SUBAPPLICATION MF (* Subapplication Type *)
  (* Standard: 61499-2 *)
  (* Version 1.0, 2025-02-12, franz *)
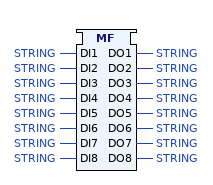
  VAR_INPUT
    DI1 : STRING;
    DI2 : STRING;
    DI3 : STRING;
    DI4 : STRING;
    DI5 : STRING;
    DI6 : STRING;
    DI7 : STRING;
    DI8 : STRING;
  END_VAR
  VAR_OUTPUT
    DO1 : STRING;
    DO2 : STRING;
    DO3 : STRING;
    DO4 : STRING;
    DO5 : STRING;
    DO6 : STRING;
    DO7 : STRING;
    DO8 : STRING;
  END_VAR
END_SUBAPPLICATION
